// TIA Portal V18 program export: 1 tag tables, 0 data types, 1 data blocks, 4 code blocks (in call order from the OBs), 2 instance data blocks

VAR_GLOBAL   // PLC tag table "Standard-Variablentabelle"
   start AT %I0.0 : Bool;
   stop AT %I0.1 : Bool;
   drain AT %I0.2 : Bool;
   levelMeter AT %ID30 : Real;
   SetPoint AT %ID38 : Real;
   FillValve AT %QD30 : Real;
   DissValve AT %QD34 : Real;
   SetPointDisplay AT %QD38 : DInt;
   LevelDisplay AT %QD42 : DInt;
   ErrorDisplay AT %QD46 : Real;
   Tag_1 AT %M0.0 : Bool;
   Tag_2 AT %MD100 : Real;
   scaledlevel AT %MW2 : Int;
   setscaled AT %MW12 : Int;
   Tag_3 AT %M2.2 : Bool;
END_VAR

DATA_BLOCK "hmi"   // DB5
{ S7_Optimized_Access := 'TRUE' }
VERSION : 0.1
// stored: AutoNumber true, IsOnlyStoredInLoadMemory false, IsRetainMemResEnabled false, IsWriteProtectedInAS false, MemoryReserve 100
   VAR
      startfromhmi : Bool;
   END_VAR
BEGIN
END_DATA_BLOCK

ORGANIZATION_BLOCK "Main"   // OB1, LAD, ProgramCycle
TITLE = "Main Program Sweep (Cycle)"
{ S7_Optimized_Access := 'TRUE' }
VERSION : 0.1
// stored: AutoNumber true, IsIECCheckEnabled false, SetENOAutomatically false
   VAR_INPUT
      Initial_Call : Bool;   // Initial call of this OB
      Remanence : Bool;   // =True, if remanent data are available
   END_VAR
   VAR_TEMP
      norm3 : Real;
   END_VAR
BEGIN

REGION Network 1: FOR FACTORY I/O
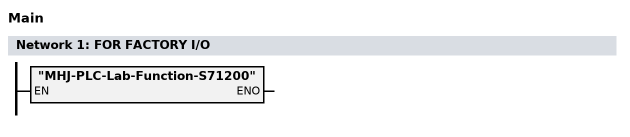
   RUNG wire#powerrail
      "MHJ-PLC-Lab-Function-S71200"()
   END_RUNG
   // the same network as SCL:
   "MHJ-PLC-Lab-Function-S71200"();
END_REGION
END_ORGANIZATION_BLOCK

FUNCTION "MHJ-PLC-Lab-Function-S71200" : Void   // FC9000, SCL
{ S7_Optimized_Access := 'TRUE' }
VERSION : 0.1
// stored: AutoNumber false, IsIECCheckEnabled false, SetENOAutomatically false, UDAEnableTagReadback false
   VAR_TEMP
      rdTimeReturn : Int;
      outputTime : DTL;
      SyncVal : Byte;
      forVal : Int;
      forVal_2 : Int;
      Value : Byte;
   END_VAR
   VAR CONSTANT
      CompVal : Byte := 16#34;
      Value_01 : Byte := 16#11;
      Value_01_DW : DWord := 16#A165_D992;
      Value_02_DW : DWord := 16#58BE_4401;
   END_VAR
BEGIN

   #Value:=PEEK(area := 16#82,
        dbNumber := 0,
        byteOffset := 511);
   #Value := #Value + 1;

   POKE(area := 16#82,
        dbNumber := 0,
        byteOffset := 511,
        value := #Value);

   POKE(area:=16#81,
        dbNumber:=0,
        byteOffset:=1016,
        value:=#Value_01_DW);
   POKE(area := 16#81,
        dbNumber := 0,
        byteOffset := 1020,
        value := #Value_02_DW);

   POKE(area := 16#81,
        dbNumber := 0,
        byteOffset := 511,
        value := B#16#00);

   FOR #forVal := 0 TO 120 DO
       FOR #forVal_2:=0 TO 10 DO
           #rdTimeReturn:=RD_SYS_T(#outputTime);
           #rdTimeReturn := WR_SYS_T(#outputTime);
           #rdTimeReturn := RD_SYS_T(#outputTime);
           #rdTimeReturn := WR_SYS_T(#outputTime);
       END_FOR;
       #SyncVal:= PEEK(area := 16#81,
                      dbNumber := 0,
                      byteOffset := 511);
       IF #SyncVal = #CompVal THEN
          GOTO M_1;
       END_IF;
   END_FOR;
   RETURN;

   M_1:
   POKE(area := 16#81,
        dbNumber := 0,
        byteOffset := 511,
        value := B#16#0);
END_FUNCTION

ORGANIZATION_BLOCK "Cyclic interrupt"   // OB30, LAD, CyclicInterrupt
{ S7_Optimized_Access := 'TRUE' }
VERSION : 0.1
// stored: AutoNumber true, IsIECCheckEnabled false, SetENOAutomatically false
   VAR_INPUT
      Initial_Call : Bool;   // Initial call of this OB
      Event_Count : Int;   // Events discarded
   END_VAR
BEGIN

REGION Network 1
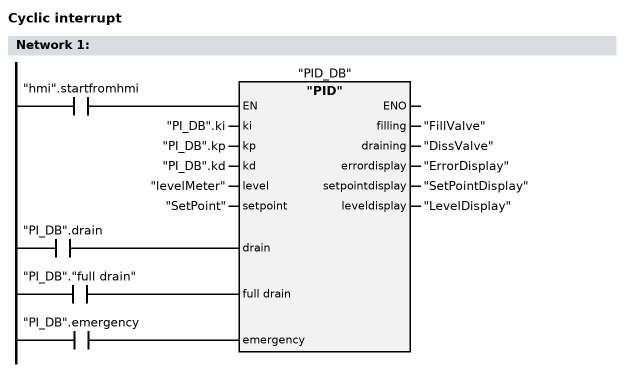
   RUNG wire#powerrail
      Contact( "hmi".startfromhmi )
      "PID_DB"(drain := wire#w1, "full drain" := wire#w2, emergency := wire#w3, ki := "PI_DB".ki, kp := "PI_DB".kp, kd := "PI_DB".kd, level := "levelMeter", setpoint := "SetPoint", filling => "FillValve", draining => "DissValve", errordisplay => "ErrorDisplay", setpointdisplay => "SetPointDisplay", leveldisplay => "LevelDisplay")
   END_RUNG
   RUNG wire#powerrail
      Contact( "PI_DB".drain )
   END_RUNG wire#w1
   RUNG wire#powerrail
      Contact( "PI_DB"."full drain" )
   END_RUNG wire#w2
   RUNG wire#powerrail
      Contact( "PI_DB".emergency )
   END_RUNG wire#w3
   // the same network as SCL:
   IF "hmi".startfromhmi THEN
       "PID_DB"(ki := "PI_DB".ki,   // "PID"
                kp := "PI_DB".kp,
                kd := "PI_DB".kd,
                level := "levelMeter",
                setpoint := "SetPoint",
                drain := "PI_DB".drain,
                "full drain" := "PI_DB"."full drain",
                emergency := "PI_DB".emergency,
                filling => "FillValve",
                draining => "DissValve",
                errordisplay => "ErrorDisplay",
                setpointdisplay => "SetPointDisplay",
                leveldisplay => "LevelDisplay");
   END_IF;
END_REGION

REGION Network 2 (SCL): TO BE SURE THAT KP ON PID WILL BE ALWAYS BIGGER THAN 1
   IF "PI_DB".kp < 1 THEN
       "PI_DB".kp := 1;
   END_IF;
END_REGION
END_ORGANIZATION_BLOCK

FUNCTION_BLOCK "PID"   // FB1, SCL
{ S7_Optimized_Access := 'TRUE' }
VERSION : 0.1
// stored: AutoNumber true, IsIECCheckEnabled false, IsRetainMemResEnabled false, MemoryReserve 100, SetENOAutomatically false, UDAEnableTagReadback false
   VAR_INPUT
      ki : Real := 0.002;
      kp : Real := 11.0;
      kd : Real;
      level : Real;
      setpoint : Real;
      drain : Bool;
      "full drain" : Bool;
      emergency : Bool;
   END_VAR
   VAR_OUTPUT
      filling : Real;
      draining : Real;
      errordisplay : Real;
      setpointdisplay : DInt;
      leveldisplay : DInt;
   END_VAR
   VAR
      integralop : Real;
      oldintegral : Real;
      err2 : Real;
   END_VAR
   VAR_TEMP
      error : Real;
      u : Real;
      temp : DInt;
   END_VAR
BEGIN

   #errordisplay := ABS(#setpoint - #level);

   //display setpoint to 100%
   #setpointdisplay := REAL_TO_DINT(#setpoint*10.0);
   //



   //display level to 100%
   #leveldisplay :=REAL_TO_DINT( #level*10.0);
   //
   #temp := REAL_TO_DINT(#kp);

   #error := #setpoint - #level;

   #integralop := #integralop + #error; //sums all the past errors to present error
   #u := (#error * #kp) + (#integralop * (#ki / 10)) + (#kd * (#err2 - #error));
   #filling := #u;
   #draining := -#u;


   //if error always goes up the filling will always goes up
   //and it will be more that 100% .but the valve can go only to 100% open
   //so if it goes up.we stop the valve at 10 and  stabilized the integral
   IF (#filling > 10.0) THEN
       #integralop := #oldintegral;
       #filling := 10.0;
   END_IF;
   //same thing but for values under 0
   IF (#filling < 0.0) THEN
       #integralop := #oldintegral;
       #filling := 0.0;
   END_IF;
   IF (#draining > 10.0) THEN
       #integralop := #oldintegral;
       #draining := 10.0;
   END_IF;

   IF (#draining < 0.0) THEN
       #integralop := #oldintegral;
       #draining := 0.0;
   END_IF;

   #oldintegral := #integralop; //past error sum
   #err2 := #error;//past error

   IF #drain THEN
       #draining := 10.0;

   END_IF;

   IF #"full drain" THEN
       #draining := 10.0;
       #filling := 0;
   END_IF;
   IF #emergency THEN
       #draining := 0;
       #filling := 0;

   END_IF;
END_FUNCTION_BLOCK

DATA_BLOCK "PID_DB"   // DB6
VERSION : 0.1
// stored: AutoNumber true, InstanceOfName PID, InstanceOfType FB
"PID"
BEGIN
END_DATA_BLOCK

DATA_BLOCK "PI_DB"   // DB3
VERSION : 0.1
// stored: AutoNumber true, InstanceOfName PID, InstanceOfType FB
"PID"
BEGIN
END_DATA_BLOCK
